{attribute addProperty BoxType "EL6201-0000-0017"}
{attribute addProperty Id "Slave_8A_DO0BIT10.12557Slave_8A_DO1BIT10.12558Slave_8A_DO2BIT10.12559Slave_8A_DO3BIT10.12560Slave_8B_DO0BIT10.12561Slave_8B_DO1BIT10.12562Slave_8B_DO2BIT10.12563Slave_8B_DO3BIT10.12564"}
{attribute addProperty CRC "3377216482"}
{attribute addProperty SizeInBites "8"}
{attribute addProperty SizeInBytes "1"}
TYPE Slave_8_Outputs_C94C3BE2 :
STRUCT
	{attribute addProperty Name "Slave_8A_DO0"}
	Slave_8A_DO0 : BIT;
	{attribute addProperty Name "Slave_8A_DO1"}
	Slave_8A_DO1 : BIT;
	{attribute addProperty Name "Slave_8A_DO2"}
	Slave_8A_DO2 : BIT;
	{attribute addProperty Name "Slave_8A_DO3"}
	Slave_8A_DO3 : BIT;
	{attribute addProperty Name "Slave_8B_DO0"}
	Slave_8B_DO0 : BIT;
	{attribute addProperty Name "Slave_8B_DO1"}
	Slave_8B_DO1 : BIT;
	{attribute addProperty Name "Slave_8B_DO2"}
	Slave_8B_DO2 : BIT;
	{attribute addProperty Name "Slave_8B_DO3"}
	Slave_8B_DO3 : BIT;
END_STRUCT
END_TYPE

(* stored: Version 1.2.0.0, ProductVersion 3.1.4024.9
   DUT Slave_8_Outputs_C94C3BE2: Id {19523e9c-9acc-48da-a8f4-6c2dc87a8b21} *)
